// TIA Portal V18 export
// export: Created 2025-12-01T17:53:04.5110192Z, ExportSetting None, DisplayName Totally Integrated Automation Portal, DisplayVersion V18 Update 5, DisplayName TIA Portal Openness, DisplayVersion V18 Update 5, DisplayName TIA Portal Teamcenter Gateway, DisplayVersion V18, DisplayName TIA Portal Version Control Interface, DisplayVersion V18, DisplayName STEP 7 Professional, DisplayVersion V18 Update 5, DisplayName STEP 7 Safety, DisplayVersion V18, DisplayName WinCC Professional, DisplayVersion V18 Update 5
Screen "270_Cylinder_J1"  1280x800, Number=270, Template=02ManualUnit1
  ScreenLayer "Layer_0"
    FaceplateInstance "Cylinder_S71500_TP700_1" at 0,85 size 1279x80  FaceplateTypeName=03 FunctionBlocks@$@101 Cylinder@$@101.2 HMI@$@S7-1500@$@Cylinder_S71500_TP700 V 0.0.29
      Cy := STxxxCylinder031
      CylinderName := Cyl name
      HomeButtonName := Cyl go home button
      WorkButtonName := Cyl go work button
      HomeQaddress := Cyl home Q
      HomeIaddress := Cyl home I
      WorkIaddress := Cyl work I
      WorkQaddress := Cyl work Q
    FaceplateInstance "Cylinder_S71500_TP700_3" at 0,160 size 1279x80  FaceplateTypeName=03 FunctionBlocks@$@101 Cylinder@$@101.2 HMI@$@S7-1500@$@Cylinder_S71500_TP700 V 0.0.29
      Cy := STxxxCylinder032
      CylinderName := Cyl name
      HomeButtonName := Cyl go home button
      WorkButtonName := Cyl go work button
      HomeQaddress := Cyl home Q
      HomeIaddress := Cyl home I
      WorkIaddress := Cyl work I
      WorkQaddress := Cyl work Q
    Button "btnMenu4" at 384,725 size 128x75  TextOff="J-气缸2 / J-Cylinder2", TextOn="J-气缸2 / J-Cylinder2"
      on Click: ActivateScreen(Screen name := 273_Cylinder_J2, Object number := 0)
    Button "btnMenu5" at 512,725 size 128x75  TextOff="J-电机2 / J-Motor2", TextOn="J-电机2 / J-Motor2"
      on Click: ActivateScreen(Screen name := 274_Motor_J2, Object number := 0)
    Button "btnMenu6" at 640,725 size 128x75  TextOff="J-气缸3 / J-Cylinder3", TextOn="J-气缸3 / J-Cylinder3"
      on Click: ActivateScreen(Screen name := 276_Cylinder_J3, Object number := 0)
    Button "btnMenu7" at 896,725 size 128x75
    Button "btnMenu6_1" at 768,725 size 128x75  TextOff="J-电机3 / J-Motor3", TextOn="J-电机3 / J-Motor3"
      on Click: ActivateScreen(Screen name := 277_Motor_J3, Object number := 0)
    Button "btnMenu7_1" at 1024,725 size 128x75
    Button "按钮_9" at 128,725 size 128x75  PictureOff=向右箭头_0, TextOff="J-气缸1 / J-Cylinder1", TextOn="J-气缸1 / J-Cylinder1"
      on Click: ActivateScreen(Screen name := , Object number := 0)
    Button "btnMenu4_1" at 256,725 size 128x75  TextOff="J-电机1 / J-Motor1", TextOn="J-电机1 / J-Motor1"
      on Click: ActivateScreen(Screen name := 271_Motor_J1, Object number := 0)
    GraphicView "图形视图_1" at 98,253 size 1108x420  Picture=图形_58
